{attribute 'qualified_only'}
VAR_GLOBAL
END_VAR

(* stored: Version 1.1.0.1, ProductVersion 3.1.4024.13
   GVL GVL: Id {e9b6b1bc-3ad8-4475-b9de-9556a2800ab9} *)
